Staubli VAL3: clearScreen.pgx

public program clearScreen()
begin

  // Do nothing - not needed on CS9

end
